//{attribute 'qualified_only'}
VAR_GLOBAL
	fb_PB_ITC_ManagerConveyor 		: FB_PB_ITC_Conveyor;		
END_VAR

(* stored: Version 1.1.0.1, ProductVersion 3.1.4022.12
   GVL ProBox_Conveyor: Id {96d058ce-c565-4d52-8463-ccf132bf0a06} *)
